FUNCTION F_WSTRING_ARG : ST_Arg
VAR_INPUT
	wsInput : WSTRING(255);
END_VAR
VAR
	stArg : ST_Arg;
	sysVar_Info : __SYSTEM.VAR_INFO;
END_VAR

sysVar_Info 	:= __VARINFO(wsInput);
stArg.TypeClass := sysVar_Info.TypeClass;
stArg.pValue 	:= 0;
stArg.diSize 	:= SIZEOF(wsInput);
stArg.sValue 	:= TO_STRING(wsInput); 
F_WSTRING_ARG := stArg;

END_FUNCTION

(* stored: Version 1.1.0.1, ProductVersion 3.1.4024.4
   POU F_WSTRING_ARG: Id {6322a4b9-e84c-47ac-87d4-305c6ce01fa9}, SpecialFunc None *)
